{attribute 'qualified_only'}
{attribute 'strict'}
{attribute 'to_string'}
TYPE E_AlarmOperator :
(
	Invalid := 0,
    GreaterThan,
    LessThan,
    Equal,
    GreaterOrEqual,
    LessOrEqual
);
END_TYPE

(* stored: Version 1.1.0.1, ProductVersion 3.1.4026.18
   DUT E_AlarmOperator: Id {b76febb0-de45-4da9-aab5-388700bc550f} *)
